// TIA Portal V19 export
FUNCTION_BLOCK "SCALE"   // FB4, LAD
{ S7_Optimized_Access := 'TRUE' }
// stored: MemoryReserve 100, SetENOAutomatically false
   VAR_INPUT
      "SCALE MIN" : Real;
      "SCALE MAX" : Real;
      INPUT : Int;
      "RAW MIN" : Int;
      "RAW MAX" : Int;
   END_VAR
   VAR_OUTPUT
      "PV VALUE" : Real;
   END_VAR
   VAR_TEMP
      NORMX : Real;
   END_VAR
BEGIN

REGION Network 1
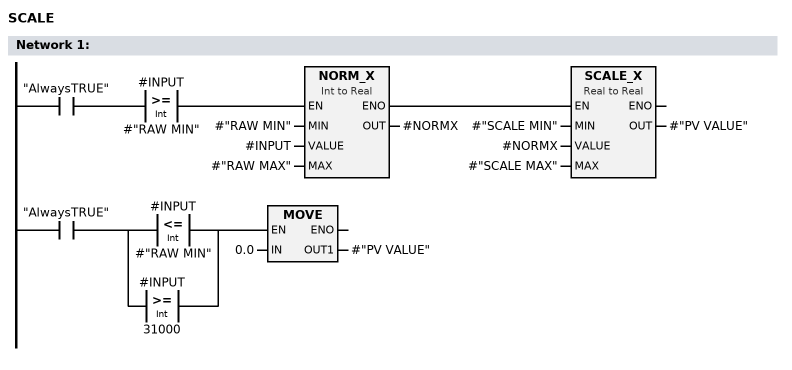
   RUNG wire#powerrail
      Contact( "AlwaysTRUE" )
      { S7_Templates := "SrcType := Int" } GE_Contact(in1 := #INPUT, in2 := #"RAW MIN")
      { S7_Templates := "[SrcType := Int, DestType := Real]" } Normalize(min := #"RAW MIN", value := #INPUT, max := #"RAW MAX", out => #NORMX)
      { S7_Templates := "[SrcType := Real, DestType := Real]" } Scale(min := #"SCALE MIN", value := #NORMX, max := #"SCALE MAX", out => #"PV VALUE")
   END_RUNG
   RUNG wire#powerrail
      Contact( "AlwaysTRUE" )
      wire#w1
      { S7_Templates := "SrcType := Int" } LE_Contact(in1 := #INPUT, in2 := #"RAW MIN")
      wire#w2
      Move(in := 0.0, out1 => #"PV VALUE")
   END_RUNG
   RUNG wire#w1
      { S7_Templates := "SrcType := Int" } GE_Contact(in1 := #INPUT, in2 := 31000)
   END_RUNG wire#w2
   // the same network as SCL:
   IF "AlwaysTRUE" AND (#INPUT >= #"RAW MIN") THEN
       #NORMX := NORM_X(MIN := #"RAW MIN", VALUE := #INPUT, MAX := #"RAW MAX");
       #"PV VALUE" := SCALE_X(MIN := #"SCALE MIN", VALUE := #NORMX, MAX := #"SCALE MAX");
   END_IF;
   IF "AlwaysTRUE" AND ((#INPUT <= #"RAW MIN") OR (#INPUT >= 31000)) THEN #"PV VALUE" := 0.0; END_IF;
END_REGION
END_FUNCTION_BLOCK
